// TIA Portal V17 export
// export: Created 2024-09-02T12:50:12.4997885Z, ExportSetting WithDefaults, DisplayName Totally Integrated Automation Portal, DisplayVersion V17, DisplayName TIA Portal Openness, DisplayVersion V17, DisplayName TIA Portal Version Control Interface, DisplayVersion V17, DisplayName STEP 7 Professional, DisplayVersion V17, DisplayName STEP 7 Safety, DisplayVersion V17, DisplayName WinCC Professional, DisplayVersion V17
FUNCTION "AnwFC_Process_FG02_BEA_OP70" : Void   // FC501, LAD
TITLE = Process / Prozess
{ S7_Optimized_Access := 'TRUE' }
AUTHOR : VAF
FAMILY : PROZESS
NAME : PROZESS
VERSION : 0.1
// stored: AutoNumber false, IsIECCheckEnabled false, SetENOAutomatically false, UDAEnableTagReadback false
BEGIN

REGION Network 1: Processing dates 1 / Bearbeitungsdaten 1
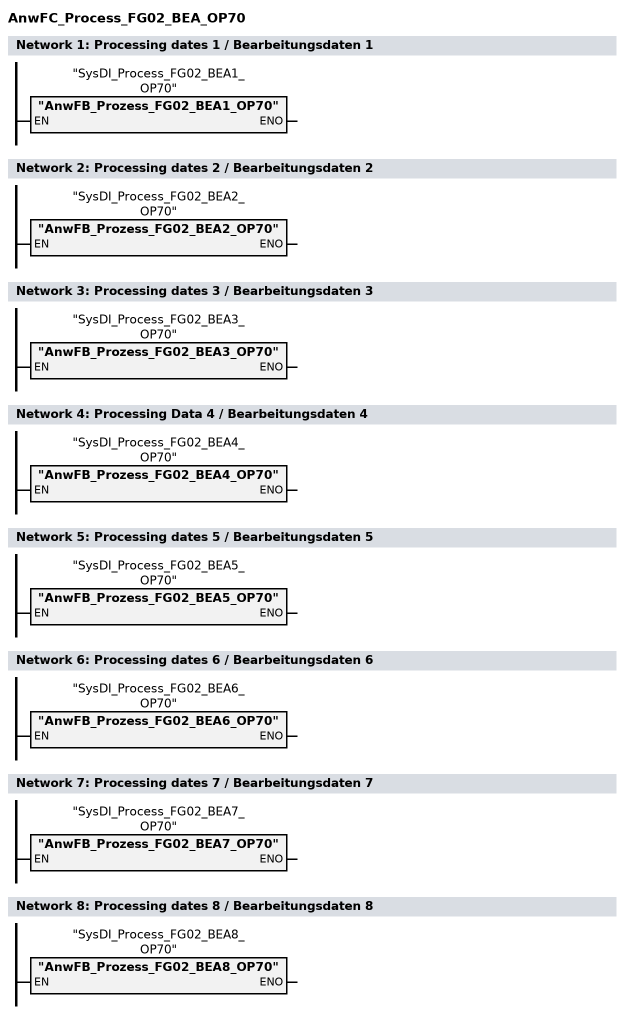
   RUNG wire#powerrail
      "SysDI_Process_FG02_BEA1_OP70"()
   END_RUNG
   // the same network as SCL:
   "SysDI_Process_FG02_BEA1_OP70"();   // "AnwFB_Prozess_FG02_BEA1_OP70"
END_REGION

REGION Network 2: Processing dates 2 / Bearbeitungsdaten 2
   RUNG wire#powerrail
      "SysDI_Process_FG02_BEA2_OP70"()
   END_RUNG
   // the same network as SCL:
   "SysDI_Process_FG02_BEA2_OP70"();   // "AnwFB_Prozess_FG02_BEA2_OP70"
END_REGION

REGION Network 3: Processing dates 3 / Bearbeitungsdaten 3
   RUNG wire#powerrail
      "SysDI_Process_FG02_BEA3_OP70"()
   END_RUNG
   // the same network as SCL:
   "SysDI_Process_FG02_BEA3_OP70"();   // "AnwFB_Prozess_FG02_BEA3_OP70"
END_REGION

REGION Network 4: Processing Data 4 / Bearbeitungsdaten 4
   RUNG wire#powerrail
      "SysDI_Process_FG02_BEA4_OP70"()
   END_RUNG
   // the same network as SCL:
   "SysDI_Process_FG02_BEA4_OP70"();   // "AnwFB_Prozess_FG02_BEA4_OP70"
END_REGION

REGION Network 5: Processing dates 5 / Bearbeitungsdaten 5
   RUNG wire#powerrail
      "SysDI_Process_FG02_BEA5_OP70"()
   END_RUNG
   // the same network as SCL:
   "SysDI_Process_FG02_BEA5_OP70"();   // "AnwFB_Prozess_FG02_BEA5_OP70"
END_REGION

REGION Network 6: Processing dates 6 / Bearbeitungsdaten 6
   RUNG wire#powerrail
      "SysDI_Process_FG02_BEA6_OP70"()
   END_RUNG
   // the same network as SCL:
   "SysDI_Process_FG02_BEA6_OP70"();   // "AnwFB_Prozess_FG02_BEA6_OP70"
END_REGION

REGION Network 7: Processing dates 7 / Bearbeitungsdaten 7
   RUNG wire#powerrail
      "SysDI_Process_FG02_BEA7_OP70"()
   END_RUNG
   // the same network as SCL:
   "SysDI_Process_FG02_BEA7_OP70"();   // "AnwFB_Prozess_FG02_BEA7_OP70"
END_REGION

REGION Network 8: Processing dates 8 / Bearbeitungsdaten 8
   RUNG wire#powerrail
      "SysDI_Process_FG02_BEA8_OP70"()
   END_RUNG
   // the same network as SCL:
   "SysDI_Process_FG02_BEA8_OP70"();   // "AnwFB_Prozess_FG02_BEA8_OP70"
END_REGION
END_FUNCTION
